{attribute 'no_explicit_call' := 'Do not call the body - Stick to OOP'}
FUNCTION_BLOCK FB_XTS_Station EXTENDS FB_CH_Object IMPLEMENTS I_XTS_Station, I_XTS_Station_PLC
VAR
	{attribute 'hide'}
	bInitDone : BOOL;
	{attribute 'hide'}
	bErrorDuringFbInit : BOOL; // Not possible to reset
	{attribute 'hide'}
	ipXtsSystem 				: I_XTS_System_Registration;
	{attribute 'hide'}	
	ipStationInFront 			: I_XTS_Station;
	{attribute 'hide'}	
	ipStationBehinde 			: I_XTS_Station;
	{attribute 'hide'}
	bSuppressDynamicsChange		: BOOL; // Suppress to change the dynamic(Gap+velocity) of passing movers. This is usefull in startup
	{attribute 'hide'}
	fMoverGapAtExit 			: LREAL; // Every mover that leaves or passes the station gets this new gap as a target.
	{attribute 'hide'}
	fMoverVelocityAtExit		: LREAL; // Every mover that leaves or passes the station gets this new velo as a target.	 
	{attribute 'hide'}
	fPositionOnTrack 			: LREAL;
	{attribute 'hide'}
	nMoverQueueSize 			: UINT;
	{attribute 'hide'}
	bReadyToRecvMovers 			: BOOL := TRUE;;
	{attribute 'hide'}
	fTargetPosWindow			: LREAL := 0.05; //[mm]
	{attribute 'hide'}
	tTargetPosMonitoringTime	: TIME := T#0MS;
	{attribute 'hide'}	
	fTrackLentgh 				: LREAL; //[mm]  Modulo
	{attribute 'hide'}
	fbAssignedMovers 			: CHALET_BaseComponents.FB_CH_List;		// List of movers approaching the station
	{attribute 'hide'}
	fbFeedback 					: CHALET_BaseComponents.FB_CH_Feedback(ipSourceInfo := fbSourceInfo);
	{attribute 'hide'}	
	bMoversInPlace : BOOL;
	
	{attribute 'TcInitSymbol'}
	OIDStationInfo : OTCID; //OID of XtsStationInfo object to visualize in Viewer. 0 if not used.
	{attribute 'hide'}
	ipStationInfo : I_TcIoXtsInfoServerInfoStation;
	{attribute 'hide'}
	bUtilityStationInitDone : BOOL;
	
	//Simulation
	{attribute 'hide'}
	fSimulationProcessDuration 	: LREAL; //[s]
	{attribute 'hide'}
	sSimulationTargedStation	: STRING; //LUID of the targed station to automatic send after the duration
	
	
	// ipXtsSystem Is Not Valid at this point, call the konstruktor again in the FB_Init
	{attribute 'hide'}
	fbTrigger 					: FB_XTS_Trigger(ipXtsSystem);
	{attribute 'hide'}
	fbSortedListMoversInQueue	: FB_XTS_Zone(ipXtsSystem);
	
	//Statistic
	{attribute 'hide'}
	fMoverPerMin				: LREAL;
	
END_VAR

METHOD AddMoverToQueue : HRESULT
VAR_INPUT
	ipMover : I_XTS_Mover;
END_VAR
VAR
	ipObject : I_CH_Object;
END_VAR
//Get I_CH_Objekt of mover to put it in to a list.
IF ipMover <> 0 AND_THEN __QUERYINTERFACE(ipMover,ipObject) THEN
	//Add in List of Movers in this station
	THIS^.fbAssignedMovers.AddObject(ipObject);
	
	//Handover information in Mover
	ipMover.ParentStation := (THIS^);

	AddMoverToQueue := S_OK;
ELSE
	AddMoverToQueue := E_FAIL;;	
END_IF
END_METHOD

METHOD ChangePos : HRESULT
VAR_INPUT
	fNewPosOnTrack : LREAL;
END_VAR
VAR
	ipEachMoverInStation : I_XTS_Mover;
	fGapToFirstMoverInQueue, fTargedPos : LREAL;
	nIdx : UDINT;
END_VAR
THIS^.fbFeedback.ActiveCommand := 'ChangePos';
THIS^.fbFeedback.Busy := TRUE;

// Only small changes during system is enabled
IF THIS^.ipXtsSystem.Enabled THEN	
	
	IF fNewPosOnTrack = THIS^.PositionOnTrack THEN
		// failed - same pos
		ChangePos := S_FALSE;
		THIS^.fbFeedback.HR := ChangePos;
		RETURN;
	END_IF	


	// new Position not allowed
	IF fNewPosOnTrack > THIS^.fTrackLentgh THEN
		// failed
		ChangePos := E_FAIL;
		THIS^.fbFeedback.HR := ChangePos;
		RETURN;
	END_IF	
	IF fNewPosOnTrack < 0 THEN
		// failed
		ChangePos := E_FAIL;
		THIS^.fbFeedback.HR := ChangePos;
		RETURN;
	END_IF	
	
	
	IF THIS^.StationBehinde <> 0 AND_THEN fNewPosOnTrack <= THIS^.StationBehinde.PositionOnTrack THEN
		// failed
		ChangePos := E_FAIL;
		THIS^.fbFeedback.HR := ChangePos;
		RETURN;
	END_IF
	IF THIS^.StationsAhead <> 0 AND_THEN fNewPosOnTrack >= THIS^.StationsAhead.PositionOnTrack THEN
		// failed
		ChangePos := E_FAIL;
		THIS^.fbFeedback.HR := ChangePos;
		RETURN;
	END_IF

	
	

	THIS^.fPositionOnTrack := fNewPosOnTrack;
	
	fbTrigger.PositionOnTrack := THIS^.fPositionOnTrack;
	
	// Move the zone 10mm forward to make sure, that an Mover who is enabled at x.01mm is still in range
	fbSortedListMoversInQueue.EndPositionOnTrack := LMOD(lr_Value:=(THIS^.PositionOnTrack + 10.0), lr_Arg:= THIS^.fTrackLentgh); 
	//The zone window is the full system, with one small exception, a window of 0.001mm after the end.  Start and end must not be identical
	fbSortedListMoversInQueue.StartPositionOnTrack := LMOD(lr_Value:=(fbSortedListMoversInQueue.EndPositionOnTrack  + 0.0001), lr_Arg:= THIS^.fTrackLentgh); 
	
	//Redo drawing of station is visu
	THIS^.bUtilityStationInitDone := FALSE;
	
	//Send all movers in this station to new position
	FOR nIdx := 0 TO (XtsParameterlist.MAX_MOVER_PER_SYSTEM-1) DO
		IF ToMover(THIS^.MoversInQueue[nIdx], ipEachMoverInStation) THEN 	
			fTargedPos := fNewPosOnTrack - fGapToFirstMoverInQueue;
			IF fTargedPos < 0 THEN
				fTargedPos := fTargedPos + THIS^.fTrackLentgh;
			END_IF
			ipEachMoverInStation.MoveAbsCA(	fPosition := fTargedPos,
											fVelocity := ipEachMoverInStation.LastCmdTargedVelocity,
											fGap	  := ipEachMoverInStation.LastCmdTargedGap,
											eDirection:= Tc3_Mc3Definitions.MC_DIRECTION.mcDirectionShortestWay	);
											
			fGapToFirstMoverInQueue := fGapToFirstMoverInQueue + ipEachMoverInStation.LastCmdTargedGap;

		ELSE
			EXIT;			
		END_IF
	END_FOR
	
	
	ChangePos := S_OK;


	
// If disabled its allowed to move to any position
ELSIF THIS^.ipXtsSystem.Disabled THEN
	THIS^.fPositionOnTrack := fNewPosOnTrack;
	ChangePos := S_OK;
	
	
	
// During disabling or enabling its not allowed to move the position	
ELSE 
	ChangePos := E_FAIL;;	
END_IF

THIS^.fbFeedback.HR := ChangePos;
END_METHOD

METHOD PROTECTED CheckForStationsSameName : HRESULT
VAR
	fbStationsToCheck : CHALET_BaseComponents.FB_CH_List;
	ipStationToCheck : I_XTS_Station;
END_VAR
VAR_INST
	{attribute 'hide'}	
	fbAlarm : FB_TcAlarm;
END_VAR
//Check for stations on the same position
fbStationsToCheck.Duplicate(THIS^.ipXtsSystem.Stations);

//Clear alarm
fbAlarm.Clear(0,0);

//Remove this station from list
fbStationsToCheck.RemoveObject(THIS^);

// go through the list and search the station in front
fbStationsToCheck.ResetIterator();
WHILE fbStationsToCheck.HasNextObject() DO
	IF ToStation(fbStationsToCheck.GetNextObject(), ipStationToCheck) THEN
		IF ipStationToCheck.PositionOnTrack = THIS^.PositionOnTrack THEN
			fbAlarm.CreateEx(stEventEntry:=TC_EVENTS.CHALET_XTS_Events.DublicateStationNames, ipSourceInfo := THIS^.fbSourceInfo, bWithConfirmation := FALSE);
			fbAlarm.ipArguments.AddStringByValue(THIS^.LUID);
			fbAlarm.Raise(0);
			CheckForStationsSameName := E_FAIL;
			RETURN;
		END_IF	
	END_IF
END_WHILE
END_METHOD

METHOD PROTECTED CheckForStationsSamePos : HRESULT
VAR
	fbStationsToCheck : CHALET_BaseComponents.FB_CH_List;
	ipStationToCheck : I_XTS_Station;
END_VAR
VAR_INST
	{attribute 'hide'}	
	fbAlarm : FB_TcAlarm;
END_VAR
//Check for stations on the same position
fbStationsToCheck.Duplicate(THIS^.ipXtsSystem.Stations);

//Clear alarm
fbAlarm.Clear(0,0);

//Remove this station from list
fbStationsToCheck.RemoveObject(THIS^);

// go through the list and search the station in front
fbStationsToCheck.ResetIterator();
WHILE fbStationsToCheck.HasNextObject() DO
	IF ToStation(fbStationsToCheck.GetNextObject(), ipStationToCheck) THEN
		IF ipStationToCheck.PositionOnTrack = THIS^.PositionOnTrack THEN
			fbAlarm.CreateEx(stEventEntry:=TC_EVENTS.CHALET_XTS_Events.DublicateStationPositions, ipSourceInfo := THIS^.fbSourceInfo, bWithConfirmation := FALSE);
			fbAlarm.ipArguments.AddStringByValue(THIS^.LUID).AddStringByValue(ipStationToCheck.LUID);
			fbAlarm.Raise(0);
			CheckForStationsSamePos := E_FAIL;
			RETURN;
		END_IF	
	END_IF
END_WHILE
END_METHOD

//Call this Methode whith seq 0->99, and wait each step until S_OK is returned
METHOD Configure : HRESULT
VAR_INPUT
	nSeq : UINT; //0->100
END_VAR
VAR

END_VAR
VAR_INST
	{attribute 'hide'}	
	fbInvalideStationPositionAlarm : FB_TcAlarm;
END_VAR
CASE nSeq OF

	1: // Reset Config-Errors
		fbInvalideStationPositionAlarm.Clear(0,0);
		

	2: //Check for valide Data
		IF 	THIS^.ipXtsSystem = 0 OR 
			THIS^.ipXtsSystem.Environment = 0 OR
			THIS^.ipXtsSystem.Stations = 0 THEN
				Configure := E_FAIL;
		END_IF	
			
	
	3: //Store some data
		THIS^.fTrackLentgh := THIS^.ipXtsSystem.TrackLength;
		IF THIS^.fTrackLentgh <= 0 THEN
			Configure := E_FAIL;
		END_IF
		
		
	10: //Station position on track is larger than CA-Group track length
		IF THIS^.PositionOnTrack > THIS^.fTrackLentgh THEN
			fbInvalideStationPositionAlarm.CreateEx(stEventEntry:=TC_EVENTS.CHALET_XTS_Events.StationPositionLargerAsTrack, ipSourceInfo := THIS^.fbSourceInfo, bWithConfirmation := FALSE);
			fbInvalideStationPositionAlarm.Raise(0);
			Configure := E_FAIL;
		END_IF

		
	20: //Error if two stations have the same LUID
		Configure := THIS^.CheckForStationsSameName();
		
				
	30: //Error if two stations have the same position on track
		Configure := THIS^.CheckForStationsSamePos();
		
		
	40: //Get Station in Front
		Configure := THIS^.GetStationAhead();
	
			
				
	50: //Get Station in Back
		Configure := THIS^.GetStationBehinde();
			
		
	60: // Config trigger fb
		THIS^.fbTrigger.ListOfMoversToCheck := THIS^.ipXtsSystem.Movers;
		THIS^.fbTrigger.PositionOnTrack := THIS^.PositionOnTrack;
		THIS^.fbTrigger.TriggerDirection := MC_Positive_Direction;
		Configure := THIS^.fbTrigger.Initialize();		
		
	70: // Config window fb		
		// Use the zone to sort all movers in this queue depending on the distance to targed in an output array.
		// Move the zone 10mm forward to make sure, that an Mover who is enabled at x.01mm is still in range
		fbSortedListMoversInQueue.EndPositionOnTrack := LMOD(lr_Value:=(THIS^.PositionOnTrack + 10.0), lr_Arg:= THIS^.fTrackLentgh); 
		//The zone window is the full system, with one small exception, a window of 0.001mm after the end.  Start and end must not be identical
		fbSortedListMoversInQueue.StartPositionOnTrack := LMOD(lr_Value:=(fbSortedListMoversInQueue.EndPositionOnTrack  + 0.0001), lr_Arg:= THIS^.fTrackLentgh); 
		fbSortedListMoversInQueue.ListOfMoversToCheck := THIS^.fbAssignedMovers;
		Configure := THIS^.fbSortedListMoversInQueue.Initialize();	
		

		
	80: //Redo drawing of station is visu
		THIS^.bUtilityStationInitDone := FALSE;	

	100..CHALET_BaseComponents.GVL_Datatypes.cMaxUint: 
		// 100..MaxUint -> Invalide input
		Configure := E_FAIL;
		
	ELSE 
		//If an step is not defind/used return ok
		Configure := S_OK;
END_CASE
END_METHOD

{attribute 'monitoring':='call'}
PROPERTY CtsEmptySpaceInQueue : UDINT
GET
//Handle UINT Overflow
IF THIS^.fbAssignedMovers.Size >= THIS^.nMoverQueueSize THEN
	CtsEmptySpaceInQueue := 0;
ELSE 
	CtsEmptySpaceInQueue := THIS^.nMoverQueueSize - THIS^.fbAssignedMovers.Size;
END_IF
END_GET
END_PROPERTY

{attribute 'monitoring':='call'}
PROPERTY CtsMoversInQueue : UDINT
GET
CtsMoversInQueue := THIS^.fbAssignedMovers.Size;
END_GET
END_PROPERTY

METHOD DeleteMoversQueue : HRESULT
VAR
	ipTempMover : I_XTS_Mover;
END_VAR
//Delete intormation in linked mover
fbAssignedMovers.ResetIterator();
WHILE fbAssignedMovers.HasNextObject() DO
	IF ToMover(fbAssignedMovers.GetNextObject(),ipTempMover) THEN
		ipTempMover.ParentStation := 0;
	END_IF	
END_WHILE

//Clear list
THIS^.fbAssignedMovers.Clear();
DeleteMoversQueue := S_OK;
END_METHOD

METHOD FB_init : BOOL
VAR_INPUT
	bInitRetains : BOOL; // if TRUE, the retain variables are initialized (warm start / cold start)
	bInCopyCode : BOOL;  // if TRUE, the instance afterwards gets moved into the copy code (online change)
	
	ipXtsSystem 			: I_XTS_System_Registration; //Interface to XTS system object
	fPositionOnTrack 		: LREAL;	//[mm]
	sUniqueName				: STRING;	//expl.:'Loading'
	nMoverQueueSize 		: UINT;		//[cts]
	
	//Dynamik at exit of station
	fMoverGapAtExit 		: LREAL;	//[mm]
	fMoverVelocityAtExit 	: LREAL;	//[mm/s]

END_VAR
VAR_INST
	{attribute 'hide'}
	bFBInitCalledOnce : BOOL; //Do the following code once during start up and not during onlinechange
END_VAR
//Do the following code once during start up and not during onlinechange
IF NOT bFBInitCalledOnce THEN 
	
	//Regristrate object in System
	IF ipXtsSystem <> 0 THEN
		ipXtsSystem.RegisterStation(THIS^);
		THIS^.ipXtsSystem := ipXtsSystem;
	END_IF

	//"" is maybe entered in an waiting or dynamic station and the name is not important
	IF sUniqueName <> '' THEN 
		THIS^.fbSourceInfo.sName := sUniqueName;
	ELSE
		sUniqueName := THIS^.fbSourceInfo.sName;
	END_IF
	
	THIS^.fMoverGapAtExit := fMoverGapAtExit;
	THIS^.fMoverVelocityAtExit := fMoverVelocityAtExit;
	THIS^.nMoverQueueSize := nMoverQueueSize;
	THIS^.fPositionOnTrack := fPositionOnTrack;
	
	THIS^.fbTrigger.FB_init(FALSE,FALSE, ipXtsSystem);
	THIS^.fbSortedListMoversInQueue.FB_init(FALSE,FALSE, ipXtsSystem);

END_IF

bFBInitCalledOnce := TRUE;
END_METHOD

(*The _ PLC interface provides the user with a simplified interface for commanding between the stations. Sometimes, however, this is not enough. 
Either you get the corresponding interface with the __Queryinterface or you can get full access with this property.*)
PROPERTY FullAccess : I_XTS_Station
GET
FullAccess := (THIS^);
END_GET
END_PROPERTY

METHOD PROTECTED GetStationAhead : HRESULT
VAR
	fbStationsToCheck	: CHALET_BaseComponents.FB_CH_List;
	ipStationToCheck 	: I_XTS_Station;	
	bTrackIsRing			: BOOL;

	fTempDistBetween 	: LREAL;
	
	fFoundDistBetween 	: LREAL := CHALET_BaseComponents.GVL_Datatypes.cMaxLreal;
	ipFoundStation		: I_XTS_Station;
END_VAR
//Clear
THIS^.ipStationInFront := 0;

//get new lisat of stations
fbStationsToCheck.Duplicate(THIS^.ipXtsSystem.Stations);

bTrackIsRing := THIS^.ipXtsSystem.Environment.TrackIsRing;


//Remove this station from list
fbStationsToCheck.RemoveObject(THIS^);

// go through the list and search the station in front
fbStationsToCheck.ResetIterator();
WHILE fbStationsToCheck.HasNextObject() DO
	IF ToStation(fbStationsToCheck.GetNextObject(), ipStationToCheck) THEN
		
		IF NOT bTrackIsRing AND (ipStationToCheck.PositionOnTrack < THIS^.PositionOnTrack) THEN
			// Skip this station if behinde and not a closed loop
			CONTINUE;
		END_IF
		
		// calc distance to position in positive direction
		fTempDistBetween := F_GetDistToPosModulo(	fActualPosition := THIS^.PositionOnTrack,
													fTargedPosition := ipStationToCheck.PositionOnTrack, 
													fModulo := THIS^.fTrackLentgh);

		// check if Station is closer then last one - store
		IF fFoundDistBetween > fTempDistBetween THEN 
			fFoundDistBetween := fTempDistBetween;
			THIS^.ipStationInFront := ipStationToCheck;
		END_IF
		
	END_IF
END_WHILE
END_METHOD

METHOD PROTECTED GetStationBehinde : HRESULT
VAR
	fbStationsToCheck	: CHALET_BaseComponents.FB_CH_List;
	ipStationToCheck 	: I_XTS_Station;	

END_VAR
//Clear
THIS^.ipStationBehinde := 0;

//get new lisat of stations
fbStationsToCheck.Duplicate(THIS^.ipXtsSystem.Stations);

//Remove this station from list
fbStationsToCheck.RemoveObject(THIS^);

// go through the list and search the station in front
fbStationsToCheck.ResetIterator();
WHILE fbStationsToCheck.HasNextObject() DO
	IF ToStation(fbStationsToCheck.GetNextObject(), ipStationToCheck) THEN
		
		IF ipStationToCheck.StationsAhead.LUID = THIS^.LUID THEN
			//FOUND
			THIS^.ipStationBehinde := ipStationToCheck;
			RETURN;
		END_IF
		
	END_IF
END_WHILE
END_METHOD

{attribute 'monitoring':='call'}
PROPERTY HR : HRESULT
GET
HR := fbFeedback.hr;
END_GET
END_PROPERTY

METHOD Initialize : HRESULT
VAR
	nLoopIndex : UDINT;
	nNbOfStationsChecked : UDINT;
	//ipThisStation, ipTempStation, ipStationInFrontTemp : I_XTS_Station;
	bErrorStationInFrontNotFound, bErrorStationBehindeNotFound : BOOL;
END_VAR
VAR_INST
	//This error cannot be reset. Requires a reset cold
	{attribute 'hide'}	
	fbInitError : FB_TcAlarm;
	{attribute 'hide'}	
	fbMissingInterfaceAlarm : FB_TcAlarm;

END_VAR
fbFeedback.ActiveCommand := 'Initialize';
fbFeedback.hr := S_PENDING;	

//Check Error during FB_Init
IF THIS^.bErrorDuringFbInit THEN
	IF NOT fbInitError.bRaised THEN 
		//This error cannot be reset. Requires a reset cold
		fbInitError.CreateEx(stEventEntry:=TC_EVENTS.CHALET_Base_Events.ErrorFBinit, ipSourceInfo := THIS^.fbSourceInfo, bWithConfirmation := FALSE);
		fbInitError.Raise(0);
	END_IF
	Initialize:= E_FAIL;
	THIS^.fbFeedback.HR := Initialize;
	RETURN;
END_IF	

//Interface to System is missing
IF THIS^.ipXtsSystem = 0 THEN
	IF NOT fbMissingInterfaceAlarm.bRaised THEN 
		//This error cannot be reset. Requires a reset cold
		fbMissingInterfaceAlarm.CreateEx(stEventEntry:=TC_EVENTS.CHALET_XTS_Events.InitializationInvalideParameter, ipSourceInfo := THIS^.fbSourceInfo, bWithConfirmation := FALSE);
		fbMissingInterfaceAlarm.Raise(0);
	END_IF
	Initialize := E_FAIL;
	THIS^.fbFeedback.HR := Initialize;
	RETURN;
END_IF


IF NOT THIS^.bInitDone THEN
	
	THIS^.DeleteMoversQueue();

//	//Validate Settings - Error
//	bErrorStationInFrontNotFound := ((ipStationInFront = 0) AND THIS^.ipXtsSystem.Environment.TrackIsRing AND (THIS^.ipXtsSystem.Stations.Size > 1));
//	bErrorStationBehindeNotFound := ((ipStationBehinde = 0) AND THIS^.ipXtsSystem.Environment.TrackIsRing AND (THIS^.ipXtsSystem.Stations.Size > 1));		
//	IF (bErrorStationInFrontNotFound OR bErrorStationBehindeNotFound OR (THIS^.LUID = '') OR (fTrackLentgh <= 0) OR (fPositionOnTrack < 0.0) OR (fPositionOnTrack >= fTrackLentgh) OR (fMoverVelocityAtExit <= 0) OR (fMoverGapAtExit <= 0)) THEN
//		fbFeedback.hr := GetMostSignificant(E_FAIL, fbFeedback.hr);	
//		IF NOT fbInitError.bRaised THEN 
//			//This error cannot be reset. Requires a reset cold
//			fbInitError.CreateEx(stEventEntry:=TC_EVENTS.CHALET_XTS_Events.InitializationInvalideParameter, ipSourceInfo := THIS^.fbSourceInfo, bWithConfirmation := FALSE);
//			fbInitError.Raise(0);
//		END_IF
//	END_IF

		THIS^.fbTrigger.ListOfMoversToCheck := THIS^.ipXtsSystem.Movers;
		THIS^.fbTrigger.PositionOnTrack := THIS^.PositionOnTrack;
		THIS^.fbTrigger.TriggerDirection := MC_Positive_Direction;
		fbSortedListMoversInQueue.EndPositionOnTrack := LMOD(lr_Value:=(THIS^.PositionOnTrack + 10.0), lr_Arg:= THIS^.fTrackLentgh); 
		fbSortedListMoversInQueue.StartPositionOnTrack := LMOD(lr_Value:=(fbSortedListMoversInQueue.EndPositionOnTrack  + 0.0001), lr_Arg:= THIS^.fTrackLentgh); 
		fbSortedListMoversInQueue.ListOfMoversToCheck := THIS^.fbAssignedMovers;	
	bInitDone := TRUE;
END_IF

IF 	bInitDone THEN
	fbFeedback.hr := S_OK;	
END_IF
							
Initialize := fbFeedback.hr;
END_METHOD

{attribute 'monitoring':='call'}
//[mm] Every mover that leaves or passes the station gets this new gap as a target.
PROPERTY MoverGapAtExit : LREAL
GET
MoverGapAtExit := fMoverGapAtExit;
END_GET
SET
fMoverGapAtExit := MoverGapAtExit;
END_SET
END_PROPERTY

{attribute 'monitoring':='call'}
PROPERTY MoverPerMin : LREAL
GET
MoverPerMin := THIS^.fMoverPerMin;
END_GET
END_PROPERTY

{attribute 'monitoring':='call'}
PROPERTY MoverQueueSize : UINT
GET
MoverQueueSize := THIS^.nMoverQueueSize;
END_GET
SET
THIS^.nMoverQueueSize := MoverQueueSize;
END_SET
END_PROPERTY

{attribute 'monitoring':='call'}
PROPERTY MoversInPlace : BOOL
GET
THIS^.Prepare();//Prepare time-critical information, if not already done


MoversInPlace := bMoversInPlace;
END_GET
END_PROPERTY

{attribute 'monitoring':='call'}
PROPERTY MoversInQueue : REFERENCE TO ARRAY [0..(XtsParameterlist.MAX_MOVER_PER_SYSTEM-1)] OF I_XTS_Mover_PLC // Return a sorted list of movers in this zone. Index 0 is the mover in Front.
GET
MoversInQueue REF= THIS^.fbSortedListMoversInQueue.MoversInZone;
END_GET
END_PROPERTY

{attribute 'monitoring':='call'}
PROPERTY MoverVelocityAtExit : LREAL //[mm/s] Every mover that leaves or passes the station gets this new velocity as a target.
GET
MoverVelocityAtExit := fMoverVelocityAtExit;
END_GET
SET
fMoverVelocityAtExit := MoverVelocityAtExit;
END_SET
END_PROPERTY

PROPERTY OID : OTCID
GET
OID := THIS^.OIDStationInfo;
END_GET
END_PROPERTY

{attribute 'monitoring':='call'}
//[mm] from the beginning of the assigned track
PROPERTY PositionOnTrack : LREAL
GET
PositionOnTrack := fPositionOnTrack;
END_GET
SET
THIS^.ChangePos(PositionOnTrack);
END_SET
END_PROPERTY

(* 
	Use this Methode to calculate time sensitive date once each cycle. Example: read analog input and convert before do get Signal propertie
*)
METHOD PROTECTED Prepare : HRESULT
VAR_INST
	{attribute 'hide'}	
	nLastUpdatedCycleCount : UDINT;
END_VAR

VAR
	nLoopIndex : UINT;
	fExpectedDistanceToParent : LREAL;
	fPositionDifference : LREAL;
	nCycleTime_ms : UDINT;
	bMoverInQueue : BOOL;
	bTempMoverInPosition : BOOL;
	bTempMoverVeloZero : BOOL;
	bTempMoverInMonitoringTime : BOOL;
	bTempMoverThisStationAsTarged : BOOL;
END_VAR
VAR_INST
	{attribute 'hide'}
	nCycleCountInPos : UDINT;
END_VAR
//Check if this Cycle the dates are allready prepared. This is important for time sensitive informations.
IF nLastUpdatedCycleCount <> TwinCAT_SystemInfoVarList._TaskInfo[THIS^.TaskIndex].CycleCount THEN
	nLastUpdatedCycleCount := TwinCAT_SystemInfoVarList._TaskInfo[THIS^.TaskIndex].CycleCount ;


	(* Check if mover is in place. Time and Position window *)
	//If queuesize is zero, mover is never in place.
	IF nMoverQueueSize = 0 OR NOT ipXtsSystem.Enabled THEN
		THIS^.bMoversInPlace := FALSE;
		nCycleCountInPos := 0;
	ELSE
		//Get this task cycle Count and time 
		nCycleTime_ms := TwinCAT_SystemInfoVarList._TaskInfo[THIS^.nTaskIndex].CycleTime(*100ns*) / 10_000 ;
		
		bTempMoverInPosition := TRUE; bTempMoverVeloZero := TRUE; bTempMoverThisStationAsTarged := TRUE;
		fExpectedDistanceToParent := 0;
		FOR nLoopIndex := 0 TO (THIS^.nMoverQueueSize-1) DO
			IF THIS^.fbSortedListMoversInQueue.MoversInZone[nLoopIndex] <> 0 THEN
				//Check position and Gap - 1 mover do not have a gap
				IF nLoopIndex <> 0 THEN
					fExpectedDistanceToParent := fExpectedDistanceToParent + THIS^.fbSortedListMoversInQueue.MoversInZone[nLoopIndex].LastCmdTargedGap;
				END_IF
				bMoverInQueue		:= TRUE;
				
				fPositionDifference := F_GetDistToPosModulo(fTargedPosition := (THIS^.PositionOnTrack - fExpectedDistanceToParent),  fActualPosition :=  THIS^.fbSortedListMoversInQueue.MoversInZone[nLoopIndex].FullAccess.getAxisRef.NcToPlc.ModuloActPos, fModulo := THIS^.ipXtsSystem.TrackLength);
				IF fPositionDifference > (THIS^.ipXtsSystem.TrackLength/2) THEN
					fPositionDifference := (THIS^.ipXtsSystem.TrackLength - fPositionDifference);
				END_IF
				
				bTempMoverInPosition := bTempMoverInPosition AND (ABS(fPositionDifference) <= fTargetPosWindow );
				bTempMoverVeloZero := bTempMoverVeloZero AND (THIS^.fbSortedListMoversInQueue.MoversInZone[nLoopIndex].SetVelocity = 0);
				bTempMoverThisStationAsTarged := bTempMoverThisStationAsTarged AND ((THIS^.fbSortedListMoversInQueue.MoversInZone[nLoopIndex].TargedStation = THIS^.LUID));
			ELSE
				//Missing mover in queue
				bMoverInQueue := FALSE;
				EXIT;
			END_IF
		END_FOR
			
		//start time if mover position is ok
		IF bTempMoverInPosition  THEN
			nCycleCountInPos := nCycleCountInPos + 1;
		ELSE
			nCycleCountInPos := 0;
		END_IF
		
		bTempMoverInMonitoringTime := (UDINT_TO_TIME(nCycleCountInPos * nCycleTime_ms) >= tTargetPosMonitoringTime);
				
		THIS^.bMoversInPlace := bMoverInQueue AND bTempMoverInPosition AND bTempMoverInMonitoringTime AND bTempMoverThisStationAsTarged;// AND bTempMoverVeloZero;
	END_IF
	
	
END_IF
END_METHOD

{attribute 'monitoring':='call'}
PROPERTY ProcessSimulationActive : BOOL
GET
ProcessSimulationActive := THIS^.fSimulationProcessDuration > 0;
END_GET
END_PROPERTY

{attribute 'monitoring':='call'}
//prevent further movers from entering the station, 
//e.g. to prevent a collision. All movers that are already moving to reach this station will be stopped with a stop 
//and restarted with Ready True.
PROPERTY ReadyToRecvMovers : BOOL
GET
ReadyToRecvMovers := bReadyToRecvMovers;
END_GET
SET
VAR
	ipTempMover : I_XTS_Mover;
END_VAR
//Change to Not Ready:
IF (ReadyToRecvMovers = FALSE) AND (bReadyToRecvMovers <> ReadyToRecvMovers) THEN
	//halt all movers on the way
	fbAssignedMovers.ResetIterator();
	WHILE fbAssignedMovers.HasNextObject() DO
		IF ToMover(fbAssignedMovers.GetNextObject(),ipTempMover) THEN
			ipTempMover.HaltCA();	
		END_IF	
	END_WHILE
END_IF

//Change to Ready:
IF (ReadyToRecvMovers = TRUE) AND (bReadyToRecvMovers <> ReadyToRecvMovers) THEN
	//all movers that are on the way have probably been stopped before. when reactivated, the last move command is sent again.
	fbAssignedMovers.ResetIterator();
	WHILE fbAssignedMovers.HasNextObject() DO
		IF ToMover(fbAssignedMovers.GetNextObject(),ipTempMover) THEN
			ipTempMover.MoveAbsCA(	fPosition	:= THIS^.PositionOnTrack, 
								fVelocity 	:= ipTempMover.LastCmdTargedVelocity,  
								fGap 		:= ipTempMover.LastCmdTargedGap,  
								eDirection 	:= Tc3_Mc3Definitions.MC_DIRECTION.mcDirectionPositive);	
		END_IF	
	END_WHILE
END_IF

//Store new status
bReadyToRecvMovers := ReadyToRecvMovers;
END_SET
END_PROPERTY

METHOD SendMoversToStation : HRESULT //Send all Queued movers away by changing the targed station destination
VAR_INPUT
	sTargedStation	: STRING;
END_VAR
VAR
	nLoopIndex 		: UINT;;
	ipMover	: I_XTS_Mover;
END_VAR
//Invalide targed
IF sTargedStation = '' THEN
	SendMoversToStation := E_FAIL;
	RETURN;
END_IF

//Movers have not reached station and can not send away until complet
IF NOT THIS^.MoversInPlace THEN
	SendMoversToStation := E_FAIL;
	RETURN;
END_IF

//Send all Queued movers away by changing the targed station destination
FOR nLoopIndex := 0 TO nMoverQueueSize-1 DO
	IF THIS^.MoversInQueue[nLoopIndex] <> 0 AND_THEN __QUERYINTERFACE(THIS^.MoversInQueue[nLoopIndex],ipMover) THEN
		ipMover.TargedStation := sTargedStation;		
	END_IF
END_FOR
END_METHOD

//If a valid time (>0seconds) is set and the configured destination station exists, then the movers will be sent away automatically after this time from now on.
METHOD SimulationStart : HRESULT
VAR_INPUT
	fProcessDuration 	: LREAL; //[s]
	sTargedStation		: STRING; //LUID of the targed station to automatic send after the duration
END_VAR
VAR
	ipStation	: I_CH_Object;
	bValideLUID : BOOL;
END_VAR
//Search LUID in Stationslist
ipStation := THIS^.ipXtsSystem.Stations.FindLUID(sTargedStation);
bValideLUID := (ipStation <> 0); 

IF (fProcessDuration > 0) AND bValideLUID THEN
	//Valide config
	THIS^.fSimulationProcessDuration 	:=	fProcessDuration;
	THIS^.sSimulationTargedStation 		:=	sTargedStation;
	SimulationStart := S_OK;
ELSE
	//Simulation disabled
	THIS^.SimulationStop();
	SimulationStart := S_FALSE;
END_IF
END_METHOD

//If a valid time (>0seconds) is set and the configured destination station exists, then the movers will be sent away automatically after this time from now on.
METHOD SimulationStartEx : HRESULT
VAR_INPUT
	fProcessDuration 		: LREAL; //[s]
	ipStation				: I_Xts_Station_PLC; //unique station to automatic send after the duration
END_VAR
IF ipStation <> 0 THEN
	SimulationStartEx := THIS^.SimulationStart(fProcessDuration := fProcessDuration, sTargedStation := ipStation.LUID);

ELSE
	SimulationStartEx := S_FALSE;
END_IF
END_METHOD

METHOD SimulationStop : HRESULT
//Simulation disabled
THIS^.fSimulationProcessDuration 	:=	0;
THIS^.sSimulationTargedStation 		:=	'';
END_METHOD

{attribute 'monitoring':='call'}
PROPERTY StationBehinde : I_XTS_Station
GET
StationBehinde := ipStationBehinde;
END_GET
END_PROPERTY

{attribute 'monitoring':='call'}
PROPERTY StationsAhead : I_XTS_Station
GET
StationsAhead := ipStationInFront;
END_GET
END_PROPERTY

{attribute 'monitoring':='call'}
PROPERTY SuppressDynamicsChange : BOOL // Suppress to change the dynamic(Gap+velocity) of passing movers. This is usefull in startup
GET
SuppressDynamicsChange := bSuppressDynamicsChange;
END_GET
SET
bSuppressDynamicsChange := SuppressDynamicsChange;
END_SET
END_PROPERTY

{attribute 'monitoring':='call'}
//A time that is waited as soon as the mover is in the station (including the monitoring window) before “MoversInPlace” is set. e.g. used to stabilize the workpiece
PROPERTY TargetPosMonitoringTime : TIME
GET
TargetPosMonitoringTime := tTargetPosMonitoringTime;
END_GET
SET
tTargetPosMonitoringTime := TargetPosMonitoringTime;
END_SET
END_PROPERTY

{attribute 'monitoring':='call'}
//How many mm before the mover reaches the position is “MoversInPlace” set for the process. 
//This distance can also be set very large (e.g. 100mm) for moving past without stopping.
PROPERTY TargetPosWindow : LREAL
GET
TargetPosWindow := fTargetPosWindow;
END_GET
SET
fTargetPosWindow := TargetPosWindow;
END_SET
END_PROPERTY

//This sequence tries to transfer the mover to the next station in the direction of travel and checks whether the next station has space for it. 
//If the next station is a "dummy" that only changes the dynamics of the passing mover, this station is skipped and the next station is searched one ahead.
//If the station is fully occupied, no action is taken and a new search can be made in the next cycle.
METHOD PROTECTED TrySendMoverToNextStation : HRESULT
VAR_INPUT
	ipMover	: I_XTS_Mover;
	fVelocity : LREAL;
	fGap : LREAL;
END_VAR
VAR
	bStationIsOnlyForDynamicChanges : BOOL;
	bStationIsFull					: BOOL;
	bStationHanMoreMoverThanAllowed : BOOL;
	bStationHasAFreePlaceInQueue 	: BOOL;
	bStationIsTheTarged				: BOOL;
	bStationIsNotReadyToRecvMovers	: BOOL;
	
	ipMoverObject 		: I_CH_Object;
	ipTempStation 		: I_XTS_Station;	
	ipTargedStation 	: I_XTS_Station;

	nXpuNo 				: UINT;
	iMoverNo 			: UINT;
	stCommand 			: ST_TcIoXtsMoverCommand;	
END_VAR
//Invalide interface
IF ipMover = 0 THEN
	TrySendMoverToNextStation := E_FAIL;
	RETURN;
END_IF

//Mover is not in this Station.
IF __QUERYINTERFACE(ipMover,ipMoverObject) AND_THEN NOT THIS^.fbAssignedMovers.ObjectInList(ipMoverObject) THEN
	TrySendMoverToNextStation := E_FAIL;
	RETURN;
END_IF

//Send to actual Station is not supported
IF ipMover.TargedStation = THIS^.LUID THEN
	TrySendMoverToNextStation := E_FAIL;
	RETURN;
END_IF


ipTempStation := (THIS^);
//This sequence tries to transfer the mover to the next station in the direction of travel and checks whether the next station has space for it. 
//If the next station is a "dummy" that only changes the dynamics of the passing mover, this station is skipped and the next station is searched one ahead.
//If the station is fully occupied, no action is taken and a new search can be made in the next cycle.
WHILE (ipTargedStation=0) DO
	
	//get next station in flow direction
	ipTempStation := ipTempStation.StationsAhead;

	//All Stations around the XTS tested, Station not Found
	IF ipTempStation.LUID = THIS^.LUID THEN
		TrySendMoverToNextStation := E_FAIL;
		RETURN;
	END_IF

	bStationHanMoreMoverThanAllowed := (ipTempStation.CtsMoversInQueue > ipTempStation.MoverQueueSize); //Maybe during statup if all movers are forced to station x.	
	bStationIsFull					:= (ipTempStation.CtsEmptySpaceInQueue = 0) AND NOT (ipTempStation.MoverQueueSize = 0);
	bStationHasAFreePlaceInQueue 	:= (ipTempStation.CtsEmptySpaceInQueue > 0);
	bStationIsOnlyForDynamicChanges := (ipTempStation.MoverQueueSize = 0);
	bStationIsTheTarged				:= (ipTempStation.LUID = ipMover.TargedStation);
	bStationIsNotReadyToRecvMovers	:= ( NOT ipTempStation.ReadyToRecvMovers); 
	
	IF bStationIsFull OR bStationHanMoreMoverThanAllowed OR bStationIsNotReadyToRecvMovers THEN
		//Next Station is a valide targed but is already full.  Exit WHILE loop and try again next time.
		EXIT;
	
	ELSIF bStationHasAFreePlaceInQueue THEN
		//Next station found. Send mover to it.
		ipTargedStation := ipTempStation;
	
	ELSIF bStationIsOnlyForDynamicChanges AND bStationIsTheTarged THEN
		//ERROR. The target position is a dynamic station and can not be reached.
		TrySendMoverToNextStation := E_FAIL;
		RETURN;
		
	ELSIF bStationIsOnlyForDynamicChanges THEN
		//Repead WHILE loop and search an station more in front.
		;
	END_IF 

END_WHILE


//Requested station was found, send movers to there if it has space.
IF ipTargedStation <> 0 THEN
	//Handover Mover
	THIS^.fbAssignedMovers.RemoveObject(ipMoverObject);
	ipTargedStation.AddMoverToQueue(ipMover);
	//Start Movement
	ipMover.MoveAbsCA(
		fPosition:= ipTargedStation.PositionOnTrack, 
		fVelocity:= fVelocity, 
		fGap:= fGap, 
		eDirection:= Tc3_Mc3Definitions.MC_DIRECTION.mcDirectionPositive);
		
	//build Log Command
	stCommand.sCommandType	:= 'leaving station';
	stCommand.sStation		:= ipTargedStation.LUID;
	stCommand.sText 		:= F_BuildLogString(fPos := ipTargedStation.PositionOnTrack, fVelocity := fVelocity, fGap := fGap);

	//get Xpu Number by AxisId
	nXpuNo := ipXtsSystem.Environment.UtilityEnvirement.GetXpuNumberByAxisId(ipMover.getAxisRef.NcToPlc.AxisId);
	//get Mover Number by AxisId
	iMoverNo := ipXtsSystem.Environment.UtilityEnvirement.XpuTcIo(nXpuNo).GetMoverNumberByAxisId(ipMover.getAxisRef.NcToPlc.AxisId);
	
	//write Log Command
	ipXtsSystem.Environment.UtilityEnvirement.XpuTcIo(nXpuNo).MoverTcIo(iMoverNo).AddCommand(stCommand);
	

	
	TrySendMoverToNextStation := S_OK;	
ELSE
	//No movemnt possible, try next cycle again		
	TrySendMoverToNextStation := S_FALSE;
END_IF
END_METHOD

METHOD Update : HRESULT
VAR
	ipMover : I_XTS_Mover;
	ipThisStation : I_XTS_Station;
	fDistToNextMover : LREAL;
	fGapRequired : LREAL;
	bGapIsEnough : BOOL; //distance is large enough to start next command
END_VAR
//Force to do init befor call update
IF NOT bInitDone THEN
	THIS^.Initialize();
	RETURN;
END_IF


// Process Simulation. All functionality packed into one method for easier overwriting
THIS^.UpdateSimulation();


// If enabled start station logic
IF THIS^.ipXtsSystem.Enabled THEN
	
	ipThisStation := (THIS^);
	//Detect mover who is passing the station whitout be in queue. Adjust to new Gap+Dynamics
	IF fbTrigger.MoverDetected AND fbTrigger.MoverAtTrigger<>0 AND NOT THIS^.bSuppressDynamicsChange THEN
		//Only if not in this queue
		IF fbTrigger.MoverAtTrigger.ParentStation <> ipThisStation THEN
			fbTrigger.MoverAtTrigger.MoveAbsCA(
				fPosition:= fbTrigger.MoverAtTrigger.LastCmdTargedPosition, 
				fVelocity:= THIS^.fMoverVelocityAtExit, 
				fGap:= THIS^.fMoverGapAtExit, 
				eDirection:= Tc3_Mc3Definitions.MC_DIRECTION.mcDirectionPositive);
		END_IF
	END_IF
	
	///distance is large enough to start next command
	//This is to prevent stationary movers from having to move backwards
	IF THIS^.MoversInQueue[0] <> 0 THEN
		fDistToNextMover := F_GetDistToPosModulo(fTargedPosition:= THIS^.MoversInQueue[0].FullAccess.NextMover.PositionOnTrack, fActualPosition:= THIS^.MoversInQueue[0].PositionOnTrack, THIS^.ipXtsSystem.TrackLength);
		fGapRequired := MAX(THIS^.MoversInQueue[0].FullAccess.LastCmdTargedGap, THIS^.MoversInQueue[0].FullAccess.NextMover.LastCmdTargedGap);
		bGapIsEnough := (fDistToNextMover >= fGapRequired);
	END_IF
	
	
	//Test if the first mover is in station and send him away, if the destination is not this station
	IF __QUERYINTERFACE(THIS^.MoversInQueue[0],ipMover) AND_THEN (ipMover.TargedStation <> THIS^.LUID) AND_THEN bGapIsEnough THEN
		//IF mover is standstill in current station, send him away whit the exitVelocity, else use the in mover stored velocity
		IF (THIS^.MoversInQueue[0].PositionOnTrack = THIS^.PositionOnTrack) THEN
			THIS^.TrySendMoverToNextStation(ipMover := ipMover, fVelocity := THIS^.fMoverVelocityAtExit, fGap := THIS^.fMoverGapAtExit);
		ELSE
			THIS^.TrySendMoverToNextStation(ipMover := ipMover, fVelocity := ipMover.LastCmdTargedVelocity, fGap := ipMover.LastCmdTargedGap);
		END_IF	
      
	END_IF
END_IF


// Utility InfoStation, used in XTS Viewer. All functionality packed into one method for easier overwriting
THIS^.UpdateUtilityStation();

// Calculate statistic values like Mover/min of this station. All functionality packed into one method for easier overwriting
THIS^.UpdateStatistic();
END_METHOD

METHOD PROTECTED UpdateSimulation : HRESULT
VAR_INST
	tonSimulationDelay : TON;
END_VAR
//Automatic send mover to next station in Simulation
//If a valid time (>0seconds) is set and the configured destination station exists, then the movers will be sent away automatically after this time from now on.
tonSimulationDelay.IN 	:= THIS^.ipXtsSystem.Enabled AND THIS^.MoversInPlace AND THIS^.ProcessSimulationActive;
tonSimulationDelay.PT	:= LREAL_TO_TIME(THIS^.fSimulationProcessDuration*1000.0);
tonSimulationDelay();
IF tonSimulationDelay.Q THEN
	THIS^.SendMoversToStation(sTargedStation := THIS^.sSimulationTargedStation);
END_IF
END_METHOD

METHOD PROTECTED UpdateStatistic : HRESULT
VAR
	nCycleTime_ns : UDINT;
END_VAR
VAR_INST
	tWaitForXTS, tWaitForProcess 	: LTIME;
	nMoverPassingStation			: UINT;
END_VAR
//Validate settings. STATISTIC_AVG_PERIOD must be >0
IF NOT TIME_TO_BOOL(XtsParameterlist.STATISTIC_AVG_PERIOD) THEN
	UpdateStatistic := E_FAIL;
	RETURN;
END_IF

//Get this task cycle time
nCycleTime_ns := TwinCAT_SystemInfoVarList._TaskInfo[THIS^.nTaskIndex].CycleTime(*100ns*) * 100;


//Depending on whether the station gives the start signal to the process or not, decide which of the two times should be incremented.
IF THIS^.MoversInPlace THEN
	tWaitForProcess := tWaitForProcess + UDINT_TO_LTIME(nCycleTime_ns);
ELSE
	tWaitForXTS 	:= tWaitForXTS + UDINT_TO_LTIME(nCycleTime_ns);
END_IF


//Check for mover who is passing the station
IF THIS^.fbTrigger.MoverDetected THEN
	nMoverPassingStation := nMoverPassingStation +1;
END_IF


//Once the period is reached. Evaluate and reset
IF (tWaitForProcess + tWaitForXTS) >= TIME_TO_LTIME(XtsParameterlist.STATISTIC_AVG_PERIOD) THEN
	
	//Calculate passing mover per minute
	THIS^.fMoverPerMin := TO_LREAL(nMoverPassingStation)*TIME_TO_LREAL(TIME#1M)/TIME_TO_LREAL(XtsParameterlist.STATISTIC_AVG_PERIOD);

	
	
	tWaitForProcess	:= LTIME#0NS;
	tWaitForXTS 	:= LTIME#0NS;
	nMoverPassingStation := 0;
END_IF
END_METHOD

METHOD PROTECTED UpdateUtilityStation : HRESULT //Utility InfoStation, used in XTS Viewer. All functionality packed into one method for easier overwriting
VAR
	aStopPositionsInfoStation : ARRAY[1..Tc3_XTS_Utility.TcIoXtsEnvironmentParameterList.MaxXtsStopPositionsPerStation] OF LREAL;
	//aPartIDs : ARRAY[1..Tc3_XTS_Utility.TcIoXtsEnvironmentParameterList.MaxXtsPartsPerXpu] OF OTCID;
	fLastStopPosition 		: LREAL;
	nLoopIndex 				: UINT;	
    ipMovers 				: CHALET_BaseComponents.I_CH_List;
	ipTempMover 			: I_XTS_Mover;
	nXpuNo 					: UINT;
	nMoverNo 				: UINT;
	pObject 				: ITComObject;
	sName 					: STRING;
END_VAR


VAR_INST

	nOldMoverQueueSize 		: UINT := CHALET_BaseComponents.GVL_Datatypes.cMaxUint;
	fOldPositionOnTrack 	: LREAL;
	anBias 					: ARRAY[1..2] OF INT;
	bInverted 				: BOOL;
END_VAR
//Validate inputs
IF THIS^.OIDStationInfo = 0 OR ipXtsSystem.Environment = 0 THEN
	RETURN;
END_IF	


// Initalize
IF NOT THIS^.bUtilityStationInitDone THEN
	//Get interface to utility station belongs to this station via OID
    FOR nLoopIndex := 1 TO ipXtsSystem.Environment.UtilityEnvirement.InfoServerTcIo(1).P_InfoStationCount DO
		IF 	ipXtsSystem.Environment.UtilityEnvirement.InfoServerTcIo(1).P_InfoStationOids[nLoopIndex] = THIS^.OIDStationInfo THEN
			THIS^.ipStationInfo := ipXtsSystem.Environment.UtilityEnvirement.InfoServerTcIo(1).InfoStationTcIo(nInfoStation:= nLoopIndex);
			EXIT;
		END_IF
	END_FOR	
	
	// calculate Position Offset
	IF THIS^.ipStationInfo <> 0 THEN			
		ipMovers := ipXtsSystem.Movers;
		ipMovers.ResetIterator();
		nLoopIndex := 0;	
		WHILE ipMovers.HasNextObject() DO
			nLoopIndex := nLoopIndex + 1;
			IF ToMover(ipMovers.GetNextObject(),ipTempMover) THEN
				//get Xpu Number by AxisId
				nXpuNo := ipXtsSystem.Environment.UtilityEnvirement.GetXpuNumberByAxisId(ipTempMover.getAxisRef.NcToPlc.AxisId);
				//get Mover Number by AxisId
				nMoverNo := ipXtsSystem.Environment.UtilityEnvirement.XpuTcIo(nXpuNo).GetMoverNumberByAxisId(ipTempMover.getAxisRef.NcToPlc.AxisId);
				//calculate Bias
				anBias[nLoopIndex] := LREAL_TO_INT(ipXtsSystem.Environment.UtilityEnvirement.XpuTcIo(nXpuNo).MoverTcIo(nMoverNo).GetPositionInfo().fPartPosition - ipTempMover.getAxisRef.NcToPlc.ModuloActPos);
				IF nLoopIndex = 2 THEN
					 EXIT;
				END_IF
			END_IF
		END_WHILE
		
		// Validate bias, check for inverted direction
		IF anBias[1] <> anBias[2] THEN
			bInverted := TRUE; 
			ipMovers.ResetIterator();
			nLoopIndex := 0;	
			WHILE ipMovers.HasNextObject() DO
				nLoopIndex := nLoopIndex + 1;
				IF ToMover(ipMovers.GetNextObject(),ipTempMover) THEN
					//get Xpu Number by AxisId
					nXpuNo := ipXtsSystem.Environment.UtilityEnvirement.GetXpuNumberByAxisId(ipTempMover.getAxisRef.NcToPlc.AxisId);
					//get Mover Number by AxisId
					nMoverNo := ipXtsSystem.Environment.UtilityEnvirement.XpuTcIo(nXpuNo).GetMoverNumberByAxisId(ipTempMover.getAxisRef.NcToPlc.AxisId);
					//calculate inverted Bias
					anBias[nLoopIndex] := LREAL_TO_INT(ipXtsSystem.TrackLength - ipXtsSystem.Environment.UtilityEnvirement.XpuTcIo(nXpuNo).MoverTcIo(nMoverNo).GetPositionInfo().fPartPosition - ipTempMover.getAxisRef.NcToPlc.ModuloActPos);
					IF nLoopIndex = 2 THEN
						 EXIT;
					END_IF
				END_IF	
			END_WHILE
		END_IF
		
		//Set unique station name
		FW_ObjMgr_GetObjectInstance(oid:= THIS^.OIDStationInfo , iid:= TC_GLOBAL_IID_LIST.IID_ITComObject, pipUnk:= ADR(pObject));
		IF pObject <> 0 THEN
			sName := THIS^.LUID;
			pObject.TcSetObjectName(ADR(sName));
			pObject.TcRelease();
		END_IF

	END_IF
	
	THIS^.bUtilityStationInitDone := TRUE;
	fOldPositionOnTrack := -1;
END_IF




// Update
// Configure/draw station in viewer on change
IF (THIS^.ipStationInfo <> 0) AND (THIS^.nMoverQueueSize <> nOldMoverQueueSize OR THIS^.fPositionOnTrack <> fOldPositionOnTrack) THEN	
	nOldMoverQueueSize := THIS^.nMoverQueueSize;
	fOldPositionOnTrack := THIS^.fPositionOnTrack;
	
	THIS^.ipStationInfo.SetPartObjectIds(ipXtsSystem.Environment.UtilityEnvirement.XpuTcIo(1).P_PartOids);
	THIS^.ipStationInfo.SetIsEnabled(TRUE);

	
	// Draw stop position if gap between mover, given by station behind, is set
	IF (StationBehinde <> 0) AND (THIS^.nMoverQueueSize > 0) AND THIS^.nMoverQueueSize <= 25 THEN
		//Clear array
		MEMSET(ADR(aStopPositionsInfoStation), SIZEOF(aStopPositionsInfoStation), 0);
		//Fill array
		FOR nLoopIndex := 1 TO THIS^.nMoverQueueSize DO
			fLastStopPosition := (nLoopIndex-1)*StationBehinde.MoverGapAtExit;
			aStopPositionsInfoStation[(nLoopIndex)] := (fLastStopPosition);
		END_FOR
		IF NOT bInverted THEN
			//Start Position
			THIS^.ipStationInfo.SetStartPositionOnPart(MAX((fPositionOnTrack + anBias[1] - fLastStopPosition), 0)); ///zzz Todo. The InfoStation can not draw stations in the modulo area
			//End Pos
			THIS^.ipStationInfo.SetEndPositionOnPart(fPositionOnTrack + anBias[1]);
		ELSE
			//Start Position
			THIS^.ipStationInfo.SetStartPositionOnPart(ipXtsSystem.TrackLength - (fPositionOnTrack + anBias[1]));					
			//End Pos
			THIS^.ipStationInfo.SetEndPositionOnPart(MAX((ipXtsSystem.TrackLength - (fPositionOnTrack + anBias[1] - fLastStopPosition)), 0)); ///zzz Todo. The InfoStation can not draw stations in the modulo area
		END_IF
		//StopPositions
		THIS^.ipStationInfo.SetStopPositions(aStopPositionsInfoStation);

		//Override color if is set to transparent
		IF THIS^.ipStationInfo.GetStationColor() = 0 THEN
			THIS^.ipStationInfo.SetStationColor(nStationColor:= CHALET_BaseComponents.E_Colors_ARGB.Darkred);
		END_IF
	ELSE
		//Clear array
		MEMSET(ADR(aStopPositionsInfoStation), SIZEOF(aStopPositionsInfoStation), 0);	
		//StopPositions
		THIS^.ipStationInfo.SetStopPositions(aStopPositionsInfoStation);
		//Start Pos
		THIS^.ipStationInfo.SetStartPositionOnPart(nStartPositionOnPart := fPositionOnTrack + anBias[1]);
		//End Position
		THIS^.ipStationInfo.SetEndPositionOnPart(nEndPositionOnPart := fPositionOnTrack + anBias[1]);
	END_IF
	
	
	
	//Color Station depending on function:
	// Waitingstation green
	IF (FIND(THIS^.LUID,'wait')>0) OR (FIND(THIS^.LUID,'Wait')>0) OR (FIND(THIS^.LUID,'Warte')>0) OR (FIND(THIS^.LUID,'warte')>0) THEN
		THIS^.UtilityStationInfo.SetStationColor(nStationColor := CHALET_BaseComponents.E_Colors_ARGB.Green);
	
	// Dynamicstation blue
	ELSIF THIS^.MoverQueueSize = 0 THEN
		THIS^.UtilityStationInfo.SetStationColor(nStationColor := CHALET_BaseComponents.E_Colors_ARGB.Royalblue);	
    
	// Process station red
	ELSE
		THIS^.UtilityStationInfo.SetStationColor(nStationColor := CHALET_BaseComponents.E_Colors_ARGB.Red);			
	END_IF

END_IF
END_METHOD

{attribute 'monitoring':='call'}
PROPERTY UtilityStationInfo : I_TcIoXtsInfoServerInfoStation
GET
UtilityStationInfo := THIS^.ipStationInfo;
END_GET
END_PROPERTY

END_FUNCTION_BLOCK

(* stored: Version 1.1.0.1, ProductVersion 3.1.4024.12
   POU FB_XTS_Station: Id {9d6b0e03-4469-4d88-a76f-37a11bb6c040}, SpecialFunc None
   Folder Enabling: Id {e6c295f3-7f5f-4110-9b8a-d6ca43c039f0}
   Folder Subobject: Id {f1383c1c-9090-48e7-8744-26a97250ac35}
   Folder Interaction with process: Id {5d242633-9b66-4eba-83a0-bac9d9b6bfed}
   Folder Simulation: Id {25563c86-7664-43c8-8b7e-06f03c783680}
   Folder Statistic: Id {d6e1880e-9bfe-43c6-b777-4e8ddc68300c}
   Folder VisuStation: Id {7f46bf33-8125-413e-8140-e0f611848e95}
   Method AddMoverToQueue: Id {b433a16d-5a87-48da-ba13-9d276025098f}
   Method ChangePos: Id {a8d0c73e-3ab4-44eb-aa6f-55980ac0acc4}
   Method CheckForStationsSameName: Id {230bd660-d627-4f3c-90ad-8710765c6e59}
   Method CheckForStationsSamePos: Id {070fe2a1-eb05-4b6d-88b4-41c004e7aed9}
   Method Configure: Id {6ab6b1f4-813e-49e0-999f-b0999d531960}
   Property CtsEmptySpaceInQueue: Id {3524b89f-cf20-42dd-adc3-106b1a7b5a4d}
   Get Get: Id {47ac791f-1716-44b2-a530-a5e295057032}
   Property CtsMoversInQueue: Id {54c8c351-f1ec-42d4-bb9a-13d43b0c7e05}
   Get Get: Id {590a2c92-3a05-464b-be05-79551e760e27}
   Method DeleteMoversQueue: Id {73521400-4702-40dd-8b53-a821c06ec117}
   Method FB_init: Id {cf0b08fb-3e86-4a57-924b-16f70406eba7}
   Property FullAccess: Id {b29d6bf3-14e1-416e-ba1b-33b90933b7fd}
   Get Get: Id {d44c4c68-6141-423b-90cb-a9b847124c98}
   Method GetStationAhead: Id {0dc77708-dac3-4afb-a1c2-de54f6a9769e}
   Method GetStationBehinde: Id {f557e089-b593-403e-b829-f78d94e2df5b}
   Property HR: Id {5e56e9c0-c790-4a4f-926f-4782a3c193b0}
   Get Get: Id {34250221-01a0-41fc-97ee-968ba8070589}
   Method Initialize: Id {af230fb1-c1e6-41b1-9a0d-92e112111e41}
   Property MoverGapAtExit: Id {9b98ca17-b5cd-4307-a836-07b05bd3767e}
   Get Get: Id {5852ab5a-7490-4ca6-863f-095dd11ff6a2}
   Set Set: Id {15ded2d8-ff3f-40c4-9bfb-55929cfe328e}
   Property MoverPerMin: Id {b590ec11-69a5-44a8-960c-bfa7131b9c48}
   Get Get: Id {2978f893-c9ec-490f-a551-4e626d2bf940}
   Property MoverQueueSize: Id {9a2dffb4-75fa-45ae-800a-4086f0ba9d7d}
   Get Get: Id {d0b7c31b-76ee-41de-8e7a-5dfaf0c083a0}
   Set Set: Id {708d9c1b-c44a-4316-a89c-6d8d7759d82f}
   Property MoversInPlace: Id {60646129-0e50-467d-ab4b-df581af23796}
   Get Get: Id {3dae965e-73e1-44ca-9038-ef953422017c}
   Property MoversInQueue: Id {030f236d-0635-492c-b246-b079652a6b3f}
   Get Get: Id {ef69ee53-8a40-4d62-8e3f-f83bec7561ac}
   Property MoverVelocityAtExit: Id {38cc01db-991a-4223-aab5-325d96f72ddb}
   Get Get: Id {4525d5cf-d871-4104-aa92-fae008ae83b4}
   Set Set: Id {4540e606-3a9a-4961-bd7f-b277f31c0d01}
   Property OID: Id {f4f14d5e-ec72-48ac-9d56-f3adcef98296}
   Get Get: Id {da51abe5-c3d8-4208-ad8d-3dc41b216f51}
   Property PositionOnTrack: Id {3fb028d5-3e72-4276-b539-81a7277a303b}
   Get Get: Id {23500ca6-8ff4-4470-9704-4cc8e178f868}
   Set Set: Id {78940b1a-97a9-4b28-8e27-f45ef6f42cdd}
   Method Prepare: Id {484693e0-735f-4e7a-9994-8fc0fedb8e2d}
   Property ProcessSimulationActive: Id {64e091f5-4aea-4dc7-8289-a746b1855120}
   Get Get: Id {28a24689-f1f1-4227-a586-93dde7d117e9}
   Property ReadyToRecvMovers: Id {3a3d0414-1d69-4ffc-a2b9-dd988eeb331f}
   Get Get: Id {b5a50c84-8e27-475e-9c8c-e984b91c49fc}
   Set Set: Id {2b339c15-82ba-4163-97b4-9fb6e5d519e2}
   Method SendMoversToStation: Id {00d2d4cc-8dcb-4b6c-9141-305981f31067}
   Method SimulationStart: Id {f433c244-2ee8-4a20-9e47-e3d85c563490}
   Method SimulationStartEx: Id {830e0aee-0e8a-4430-97df-c96ae36a3d21}
   Method SimulationStop: Id {5c68d551-bd17-4c65-a0dd-55b7b342a33e}
   Property StationBehinde: Id {e69df2d6-cfe8-400d-9f36-6368b12b8308}
   Get Get: Id {9005a93a-2db7-49be-9a54-f061ee0c5207}
   Property StationsAhead: Id {d940311a-1fd0-4739-a62a-f18bb577fb5f}
   Get Get: Id {5b2e4462-ebe3-416c-be13-9525f2f84129}
   Property SuppressDynamicsChange: Id {2b94a5c3-f315-438f-b55d-bec1d1eb0fe0}
   Get Get: Id {2891516e-2fdb-4d69-ac6c-40b790576ca0}
   Set Set: Id {41d6bf00-27b0-4314-9a36-f49a3bb8ae5b}
   Property TargetPosMonitoringTime: Id {80283079-ac47-42d6-ab7a-e7483b8c6c34}
   Get Get: Id {404f312b-58ea-429f-8bf9-9675e23ba345}
   Set Set: Id {f4156fb8-1cfe-4165-b85f-d8fed73262c5}
   Property TargetPosWindow: Id {311bab40-a4ef-4afa-96ed-acec0607424b}
   Get Get: Id {7cd4f311-ed7b-4432-a844-c0f19e1b03b0}
   Set Set: Id {be57b3c7-44d6-4fda-886d-f5e07d767826}
   Method TrySendMoverToNextStation: Id {c191bacb-44f0-4866-b49e-61941819128a}
   Method Update: Id {56348e12-2852-4bc0-bea1-d1cb4bb9dc3f}
   Method UpdateSimulation: Id {5204600b-7c88-41e4-83d5-d5c55c52d7cc}
   Method UpdateStatistic: Id {15a2ea76-11bb-4663-9a6b-2488950a06ae}
   Method UpdateUtilityStation: Id {a456347b-90a7-402c-95c0-2f3b3511b238}
   Property UtilityStationInfo: Id {0b3829d7-344d-468c-bb26-d9e3868b191e}
   Get Get: Id {a878f674-d01c-4f97-b32a-6575de5c321b} *)
